{attribute 'conditionalshow'}
FUNCTION_BLOCK FB_CV_WORD_TO_ULINT
VAR_INPUT
	{attribute 'hide'}
	wInputValue_1				: WORD;								//Input value that is converted into the output value
	{attribute 'hide'}
	wInputValue_2				: WORD;								//Input value that is converted into the output value
	{attribute 'hide'}
	wInputValue_3				: WORD;								//Input value that is converted into the output value
	{attribute 'hide'}
	wInputValue_4				: WORD;								//Input value that is converted into the output value
	{attribute 'hide'}
	eByteOrderForConvert		: eByteOrder;						//Byte Format
END_VAR
VAR_OUTPUT
	{attribute 'hide'}
	uliOutputValue				: ULINT;							//Converted output value							
END_VAR
VAR
END_VAR

//Creator : Kai Ebensperger
//Company : Lynus AG
//Date : 28.04.2021
//Version : 1.0.0.0

//With this functionblock its possible to convert a certain Datatyp in a other Datatype
//The byte order can be selected between BigEndian and LittleEndian
//WORD TO ULINT
//Created for the Edge Device Lib over Modbus TCP
//Modbus TCP is WORD oriented

IF eByteOrderForConvert = eByteOrder.eBigEndian THEN
	uliOutputValue := SHL(WORD_TO_ULINT(wInputValue_1),48) + SHL(WORD_TO_ULINT(wInputValue_2),32) + SHL(WORD_TO_ULINT(wInputValue_3),16) + WORD_TO_DWORD(wInputValue_4);
ELSE
	uliOutputValue := SHL(WORD_TO_ULINT(wInputValue_4),48) + SHL(WORD_TO_ULINT(wInputValue_3),32) + SHL(WORD_TO_ULINT(wInputValue_2),16) + WORD_TO_DWORD(wInputValue_1);
END_IF

END_FUNCTION_BLOCK

(* stored: Version 1.1.0.1, ProductVersion 3.1.4024.9
   POU FB_CV_WORD_TO_ULINT: Id {40e98208-5670-4b8c-81a1-c27d7af75247}, SpecialFunc None *)
